ABB RAPID module: controlador3.mod

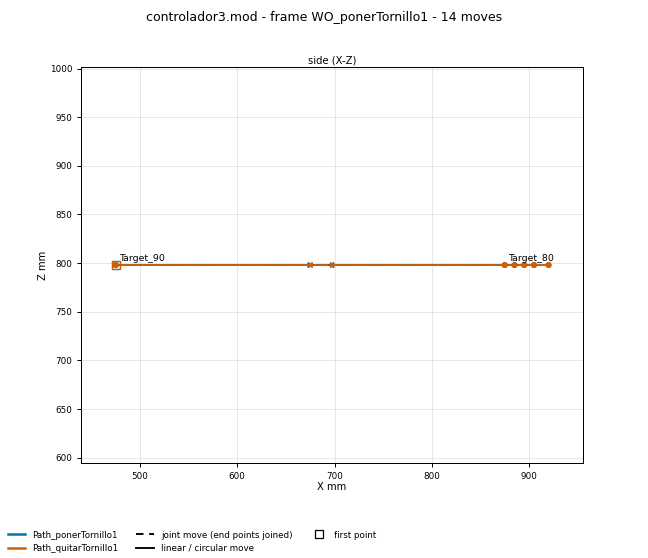
[picture p0: tool path of controlador3.mod in frame WO_ponerTornillo1, 14 of 120 moves have a stored position in this frame; points joined in program order, loops and branches not executed]
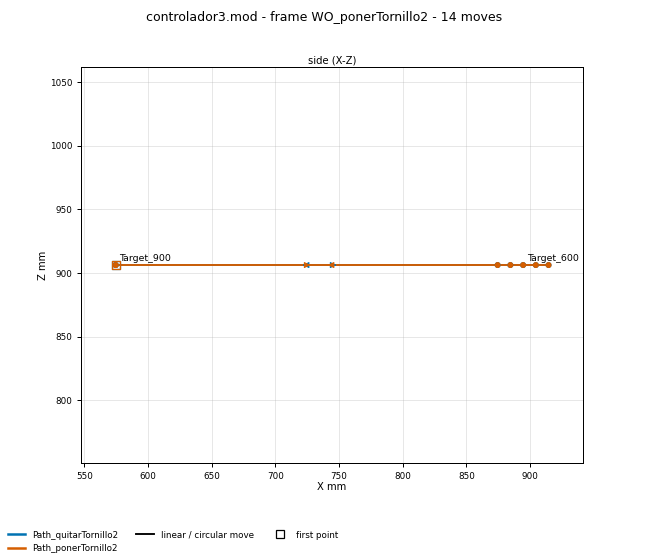
[picture p1: tool path of controlador3.mod in frame WO_ponerTornillo2, 14 of 120 moves have a stored position in this frame; points joined in program order, loops and branches not executed]
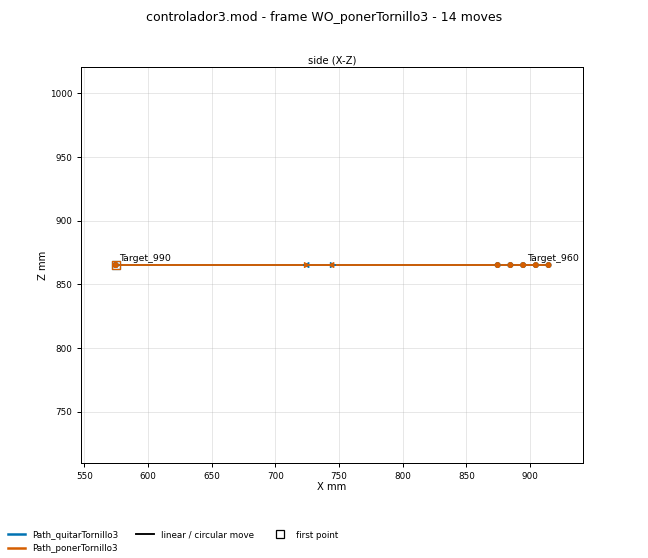
[picture p2: tool path of controlador3.mod in frame WO_ponerTornillo3, 14 of 120 moves have a stored position in this frame; points joined in program order, loops and branches not executed]
MODULE Module1
        CONST robtarget Target_30:=[[-0.058,698.771,342.903],[0,0,1,0],[1,0,1,0],[9E+09,9E+09,9E+09,9E+09,9E+09,9E+09]];
    CONST robtarget Target_20:=[[-0.058,698.771,142.903],[0,0,1,0],[1,0,1,0],[9E+09,9E+09,9E+09,9E+09,9E+09,9E+09]];
    CONST robtarget Target_10:=[[-0.058,698.771,57.903],[0,0,1,0],[0,0,0,0],[9E+09,9E+09,9E+09,9E+09,9E+09,9E+09]];
    CONST robtarget Target_40:=[[920,-282.5,798],[0.707106781,0,0.707106781,0],[-1,1,-2,0],[9E+09,9E+09,9E+09,9E+09,9E+09,9E+09]];
    CONST robtarget Target_90:=[[475,-282.5,798],[0,0.707106781,0,0.707106781],[-1,1,0,0],[9E+09,9E+09,9E+09,9E+09,9E+09,9E+09]];
    CONST robtarget Target_80:=[[875,-282.5,798],[0,0.707106781,0,0.707106781],[-1,1,0,0],[9E+09,9E+09,9E+09,9E+09,9E+09,9E+09]];
    CONST robtarget Target_70:=[[885,-282.5,798],[0.27059805,-0.653281482,0.27059805,-0.653281482],[-1,1,1,0],[9E+09,9E+09,9E+09,9E+09,9E+09,9E+09]];
    CONST robtarget Target_60:=[[895,-282.5,798],[0.5,-0.5,0.5,-0.5],[-1,1,1,0],[9E+09,9E+09,9E+09,9E+09,9E+09,9E+09]];
    CONST robtarget Target_50:=[[905,-282.5,798],[0.62578076,-0.329239185,0.62578076,-0.329239185],[-1,1,-2,0],[9E+09,9E+09,9E+09,9E+09,9E+09,9E+09]];
    CONST robtarget Target_40_1:=[[910,-282.5,798],[0.694697338,-0.131892411,0.694697338,-0.131892411],[-1,1,-2,0],[9E+09,9E+09,9E+09,9E+09,9E+09,9E+09]];
    CONST robtarget Target_55:=[[905,-282.5,798],[0.653281482,-0.27059805,0.653281482,-0.27059805],[-1,1,-2,0],[9E+09,9E+09,9E+09,9E+09,9E+09,9E+09]];
    CONST robtarget Target_45:=[[915,-282.5,798],[0.707106781,0,0.707106781,0],[-1,1,-2,0],[9E+09,9E+09,9E+09,9E+09,9E+09,9E+09]];
    CONST robtarget Target_56:=[[900,-282.5,798],[0.587937801,-0.392847479,0.587937801,-0.392847479],[-1,1,1,0],[9E+09,9E+09,9E+09,9E+09,9E+09,9E+09]];
    CONST robtarget Target_300:=[[0.2,748.407,342.618],[0,0,1,0],[0,0,0,0],[9E+09,9E+09,9E+09,9E+09,9E+09,9E+09]];
    CONST robtarget Target_200:=[[0.2,748.407,142.618],[0,0,1,0],[0,0,0,0],[9E+09,9E+09,9E+09,9E+09,9E+09,9E+09]];
    CONST robtarget Target_100:=[[0.2,748.407,57.618],[0,0,1,0],[0,0,0,0],[9E+09,9E+09,9E+09,9E+09,9E+09,9E+09]];
    CONST robtarget Target_330:=[[0.975,798.745,343.167],[0,0,1,0],[0,0,0,0],[9E+09,9E+09,9E+09,9E+09,9E+09,9E+09]];
    CONST robtarget Target_320:=[[0.975,798.745,143.167],[0,0,1,0],[0,0,0,0],[9E+09,9E+09,9E+09,9E+09,9E+09,9E+09]];
    CONST robtarget Target_310:=[[0.975,798.745,57.167],[0,0,1,0],[0,0,0,0],[9E+09,9E+09,9E+09,9E+09,9E+09,9E+09]];
    CONST robtarget Target_360:=[[0.487,848.79,342.715],[0,0,1,0],[0,0,0,0],[9E+09,9E+09,9E+09,9E+09,9E+09,9E+09]];
    CONST robtarget Target_350:=[[0.487,848.79,142.715],[0,0,1,0],[0,0,0,0],[9E+09,9E+09,9E+09,9E+09,9E+09,9E+09]];
    CONST robtarget Target_340:=[[0.487,848.79,56.715],[0,0,1,0],[0,0,0,0],[9E+09,9E+09,9E+09,9E+09,9E+09,9E+09]];
    CONST robtarget Target_390:=[[0.244,898.683,343.055],[0,0,1,0],[0,0,0,0],[9E+09,9E+09,9E+09,9E+09,9E+09,9E+09]];
    CONST robtarget Target_380:=[[0.244,898.683,143.055],[0,0,1,0],[0,0,0,0],[9E+09,9E+09,9E+09,9E+09,9E+09,9E+09]];
    CONST robtarget Target_370:=[[0.244,898.683,57.055],[0,0,1,0],[0,0,0,0],[9E+09,9E+09,9E+09,9E+09,9E+09,9E+09]];
    CONST robtarget Target_900:=[[574.529,-360.533,906.323],[0,0.707106781,0,0.707106781],[0,0,0,0],[9E+09,9E+09,9E+09,9E+09,9E+09,9E+09]];
    CONST robtarget Target_400:=[[914.529,-360.533,906.323],[0.707106781,0,0.707106781,0],[-1,1,-2,0],[9E+09,9E+09,9E+09,9E+09,9E+09,9E+09]];
    CONST robtarget Target_500:=[[904.529,-360.533,906.323],[0.653281482,-0.27059805,0.653281482,-0.27059805],[-1,1,-2,0],[9E+09,9E+09,9E+09,9E+09,9E+09,9E+09]];
    CONST robtarget Target_600:=[[894.529,-360.533,906.323],[0.5,-0.5,0.5,-0.5],[-1,1,1,0],[9E+09,9E+09,9E+09,9E+09,9E+09,9E+09]];
    CONST robtarget Target_700:=[[884.529,-360.533,906.323],[0.27059805,-0.653281482,0.27059805,-0.653281482],[-1,1,1,0],[9E+09,9E+09,9E+09,9E+09,9E+09,9E+09]];
    CONST robtarget Target_800:=[[874.529,-360.533,906.323],[0,0.707106781,0,0.707106781],[-1,1,0,0],[9E+09,9E+09,9E+09,9E+09,9E+09,9E+09]];
    CONST robtarget Target_990:=[[574.529,-487.2,865.271],[0,0.707106781,0,0.707106781],[0,0,0,0],[9E+09,9E+09,9E+09,9E+09,9E+09,9E+09]];
    CONST robtarget Target_940:=[[914.529,-487.2,865.271],[0.707106781,0,0.707106781,0],[-1,1,-2,0],[9E+09,9E+09,9E+09,9E+09,9E+09,9E+09]];
    CONST robtarget Target_950:=[[904.529,-487.2,865.271],[0.653281482,-0.27059805,0.653281482,-0.27059805],[-1,1,-2,0],[9E+09,9E+09,9E+09,9E+09,9E+09,9E+09]];
    CONST robtarget Target_960:=[[894.529,-487.2,865.271],[0.5,-0.5,0.5,-0.5],[-1,1,1,0],[9E+09,9E+09,9E+09,9E+09,9E+09,9E+09]];
    CONST robtarget Target_970:=[[884.529,-487.2,865.271],[0.27059805,-0.653281482,0.27059805,-0.653281482],[-1,1,1,0],[9E+09,9E+09,9E+09,9E+09,9E+09,9E+09]];
    CONST robtarget Target_980:=[[874.529,-487.2,865.271],[0,0.707106781,0,0.707106781],[-1,1,0,0],[9E+09,9E+09,9E+09,9E+09,9E+09,9E+09]];
    CONST robtarget Target_9000:=[[574.029,-487.592,731.451],[0,0.707106781,0,0.707106781],[0,0,0,0],[9E+09,9E+09,9E+09,9E+09,9E+09,9E+09]];
    CONST robtarget Target_4000:=[[914.029,-487.592,731.451],[0.707106781,0,0.707106781,0],[-1,1,-2,0],[9E+09,9E+09,9E+09,9E+09,9E+09,9E+09]];
    CONST robtarget Target_5000:=[[904.029,-487.592,731.451],[0.653281482,-0.27059805,0.653281482,-0.27059805],[-1,1,-2,0],[9E+09,9E+09,9E+09,9E+09,9E+09,9E+09]];
    CONST robtarget Target_6000:=[[894.029,-487.592,731.451],[0.5,-0.5,0.5,-0.5],[-1,1,1,0],[9E+09,9E+09,9E+09,9E+09,9E+09,9E+09]];
    CONST robtarget Target_7000:=[[884.029,-487.592,731.451],[0.27059805,-0.653281482,0.27059805,-0.653281482],[-1,1,1,0],[9E+09,9E+09,9E+09,9E+09,9E+09,9E+09]];
    CONST robtarget Target_8000:=[[874.029,-487.592,731.451],[0,0.707106781,0,0.707106781],[-1,1,0,0],[9E+09,9E+09,9E+09,9E+09,9E+09,9E+09]];
    CONST robtarget Target_9090:=[[574.029,-360.611,690.519],[0,0.707106781,0,0.707106781],[0,0,0,0],[9E+09,9E+09,9E+09,9E+09,9E+09,9E+09]];
    CONST robtarget Target_9040:=[[914.029,-360.611,690.519],[0.707106781,0,0.707106781,0],[-1,1,-2,0],[9E+09,9E+09,9E+09,9E+09,9E+09,9E+09]];
    CONST robtarget Target_9050:=[[904.029,-360.611,690.519],[0.653281482,-0.27059805,0.653281482,-0.27059805],[-1,1,1,0],[9E+09,9E+09,9E+09,9E+09,9E+09,9E+09]];
    CONST robtarget Target_9060:=[[894.029,-360.611,690.519],[0.5,-0.5,0.5,-0.5],[-1,1,1,0],[9E+09,9E+09,9E+09,9E+09,9E+09,9E+09]];
    CONST robtarget Target_9070:=[[884.029,-360.611,690.519],[0.27059805,-0.653281482,0.27059805,-0.653281482],[-1,1,0,0],[9E+09,9E+09,9E+09,9E+09,9E+09,9E+09]];
    CONST robtarget Target_9080:=[[874.029,-360.611,690.519],[0,0.707106781,0,0.707106781],[-1,1,0,0],[9E+09,9E+09,9E+09,9E+09,9E+09,9E+09]];
!***********************************************************
    !
    ! Módulo:  Module1
    !
    ! Descripción:
    !   <Introduzca la descripción aquí>
    !
    ! Autor: KTCHIA
    !
    ! Versión: 1.0
    !
    !***********************************************************


    !***********************************************************
    !
    ! Procedimiento Main
    !
    !   Este es el punto de entrada de su programa
    !
    !***********************************************************
    PROC main()
        !Añada aquí su código}
        SetDO Q_finish,0;
        IF E_begin=0 THEN
            WaitDI E_begin,1;
        ENDIF
        IF E_begin = 1 THEN
            SetDO Q_gripper,0;
            Path_recogerTornillo1;
            Path_ponerTornillo1;
            Path_recogerTornillo2;
            Path_ponerTornillo2;
            Path_recogerTornillo3;
            Path_ponerTornillo3;
            Path_recogerTornillo4;
            Path_ponerTornillo4;
            Path_recogerTornillo5;
            Path_ponerTornillo5;
            Path_quitarTornillo1;
            Path_descargarTornillo1;
            Path_quitarTornillo2;
            Path_descargarTornillo2;
            Path_quitarTornillo3;
            Path_descargarTornillo3;
            Path_quitarTornillo4;
            Path_descargarTornillo4;
            Path_quitarTornillo5;
            Path_descargarTornillo5;
            SetDO Q_finish,1;
        ENDIF
    ENDPROC

    PROC Path_recogerTornillo1()
        MoveJ Target_30,v500,fine,Servo\WObj:=WO_cogerTornillo1;
        SetDO Q_gripper,0;
        WaitTime 1;
        MoveL Target_20,v500,fine,Servo\WObj:=WO_cogerTornillo1;
        MoveL Target_10,v500,fine,Servo\WObj:=WO_cogerTornillo1;
        SetDO Q_gripper,1;
        WaitTime 1;
        MoveL Target_20,v500,fine,Servo\WObj:=WO_cogerTornillo1;
        MoveL Target_30,v500,fine,Servo\WObj:=WO_cogerTornillo1;
    ENDPROC
    PROC Path_ponerTornillo1()
        MoveJ Target_90,v500,fine,Servo\WObj:=WO_ponerTornillo1;
        MoveL Target_80,v500,fine,Servo\WObj:=WO_ponerTornillo1;
        MoveL Target_70,v500,fine,Servo\WObj:=WO_ponerTornillo1;
        MoveJ Target_60,v500,fine,Servo\WObj:=WO_ponerTornillo1;
        SetDO Q_gripper,0;
        WaitTime 1;
        MoveJ Target_50,v500,fine,Servo\WObj:=WO_ponerTornillo1;
        SetDO Q_gripper,1;
        WaitTime 1;
        MoveJ Target_40,v500,fine,Servo\WObj:=WO_ponerTornillo1;
        SetDO Q_gripper,0;
        WaitTime 1;
        MoveL Target_90,v500,fine,Servo\WObj:=WO_ponerTornillo1;
    ENDPROC
    PROC Path_quitarTornillo1()
        MoveJ Target_90,v500,fine,Servo\WObj:=WO_ponerTornillo1;
        MoveL Target_40,v500,fine,Servo\WObj:=WO_ponerTornillo1;
        SetDO Q_gripper,1;
        WaitTime 1;
        MoveJ Target_50,v500,fine,Servo\WObj:=WO_ponerTornillo1;
        SetDO Q_gripper,0;
        WaitTime 1;
        MoveJ Target_60,v500,fine,Servo\WObj:=WO_ponerTornillo1;
        SetDO Q_gripper,1;
        WaitTime 1;
        MoveL Target_70,v500,fine,Servo\WObj:=WO_ponerTornillo1;
        MoveL Target_80,v500,fine,Servo\WObj:=WO_ponerTornillo1;
        MoveJ Target_90,v500,fine,Servo\WObj:=WO_ponerTornillo1;
    ENDPROC
    PROC Path_descargarTornillo1()
        MoveJ Target_30,v500,fine,Servo\WObj:=WO_cogerTornillo1;
        MoveL Target_20,v500,fine,Servo\WObj:=WO_cogerTornillo1;
        MoveL Target_10,v500,fine,Servo\WObj:=WO_cogerTornillo1;
        SetDO Q_gripper,0;
        WaitTime 1;
        MoveL Target_20,v500,fine,Servo\WObj:=WO_cogerTornillo1;
        MoveL Target_30,v500,fine,Servo\WObj:=WO_cogerTornillo1;
    ENDPROC
    PROC Path_recogerTornillo2()
        SetDO Q_gripper,0;
        MoveJ Target_300,v500,fine,Servo\WObj:=WO_cogerTornillo2;
        WaitTime 1;
        MoveL Target_200,v500,fine,Servo\WObj:=WO_cogerTornillo2;
        MoveL Target_100,v500,fine,Servo\WObj:=WO_cogerTornillo2;
        SetDO Q_gripper,1;
        WaitTime 3;
        MoveL Target_200,v500,fine,Servo\WObj:=WO_cogerTornillo2;
        MoveL Target_300,v500,fine,Servo\WObj:=WO_cogerTornillo2;
    ENDPROC
    PROC Path_recogerTornillo3()
        MoveJ Target_330,v500,fine,Servo\WObj:=WO_cogerTornillo3;
        SetDO Q_gripper,0;
        WaitTime 1;
        MoveL Target_320,v500,fine,Servo\WObj:=WO_cogerTornillo3;
        MoveL Target_310,v500,fine,Servo\WObj:=WO_cogerTornillo3;
        SetDO Q_gripper,1;
        WaitTime 1;
        MoveL Target_320,v500,fine,Servo\WObj:=WO_cogerTornillo3;
        MoveL Target_330,v500,fine,Servo\WObj:=WO_cogerTornillo3;
    ENDPROC
    PROC Path_recogerTornillo4()
        MoveJ Target_360,v500,fine,Servo\WObj:=WO_cogerTornillo4;
        SetDO Q_gripper,0;
        WaitTime 1;
        MoveL Target_350,v500,fine,Servo\WObj:=WO_cogerTornillo4;
        MoveL Target_340,v500,fine,Servo\WObj:=WO_cogerTornillo4;
        SetDO Q_gripper,1;
        WaitTime 1;
        MoveL Target_350,v500,fine,Servo\WObj:=WO_cogerTornillo4;
        MoveL Target_360,v500,fine,Servo\WObj:=WO_cogerTornillo4;
    ENDPROC
    PROC Path_recogerTornillo5()
        MoveJ Target_390,v500,fine,Servo\WObj:=WO_cogerTornillo5;
        SetDO Q_gripper,0;
        WaitTime 1;
        MoveL Target_380,v500,fine,Servo\WObj:=WO_cogerTornillo5;
        MoveL Target_370,v500,fine,Servo\WObj:=WO_cogerTornillo5;
        SetDO Q_gripper,1;
        WaitTime 1;
        MoveL Target_380,v500,fine,Servo\WObj:=WO_cogerTornillo5;
        MoveL Target_390,v500,fine,Servo\WObj:=WO_cogerTornillo5;
    ENDPROC
    PROC Path_quitarTornillo2()
        MoveJ Target_900,v500,fine,Servo\WObj:=WO_ponerTornillo2;
        MoveL Target_400,v500,fine,Servo\WObj:=WO_ponerTornillo2;
        SetDO Q_gripper,1;
        WaitTime 1;
        MoveL Target_500,v500,fine,Servo\WObj:=WO_ponerTornillo2;
        SetDO Q_gripper,0;
        WaitTime 1;
        MoveL Target_600,v500,fine,Servo\WObj:=WO_ponerTornillo2;
        SetDO Q_gripper,1;
        WaitTime 1;
        MoveL Target_700,v500,fine,Servo\WObj:=WO_ponerTornillo2;
        MoveL Target_800,v500,fine,Servo\WObj:=WO_ponerTornillo2;
        MoveL Target_900,v500,fine,Servo\WObj:=WO_ponerTornillo2;
    ENDPROC
    PROC Path_quitarTornillo3()
        MoveJ Target_990,v500,fine,Servo\WObj:=WO_ponerTornillo3;
        MoveL Target_940,v500,fine,Servo\WObj:=WO_ponerTornillo3;
        SetDO Q_gripper,1;
        WaitTime 1;
        MoveL Target_950,v500,fine,Servo\WObj:=WO_ponerTornillo3;
        SetDO Q_gripper,0;
        WaitTime 1;
        MoveL Target_960,v500,fine,Servo\WObj:=WO_ponerTornillo3;
        SetDO Q_gripper,1;
        WaitTime 1;
        MoveL Target_970,v500,fine,Servo\WObj:=WO_ponerTornillo3;
        MoveL Target_980,v500,fine,Servo\WObj:=WO_ponerTornillo3;
        MoveL Target_990,v500,fine,Servo\WObj:=WO_ponerTornillo3;
    ENDPROC
    PROC Path_quitarTornillo4()
        MoveJ Target_9000,v500,fine,Servo\WObj:=WO_ponerTornillo4;
        MoveL Target_4000,v500,fine,Servo\WObj:=WO_ponerTornillo4;
        SetDO Q_gripper,1;
        WaitTime 1;
        MoveL Target_5000,v500,fine,Servo\WObj:=WO_ponerTornillo4;
        SetDO Q_gripper,0;
        WaitTime 1;
        MoveL Target_6000,v500,fine,Servo\WObj:=WO_ponerTornillo4;
        SetDO Q_gripper,1;
        WaitTime 1;
        MoveL Target_7000,v500,fine,Servo\WObj:=WO_ponerTornillo4;
        MoveL Target_8000,v500,fine,Servo\WObj:=WO_ponerTornillo4;
        MoveL Target_9000,v500,fine,Servo\WObj:=WO_ponerTornillo4;
    ENDPROC
    PROC Path_quitarTornillo5()
        MoveJ Target_9090,v500,fine,Servo\WObj:=WO_ponerTornillo5;
        MoveL Target_9040,v500,fine,Servo\WObj:=WO_ponerTornillo5;
        SetDO Q_gripper,1;
        WaitTime 1;
        MoveL Target_9050,v500,fine,Servo\WObj:=WO_ponerTornillo5;
        SetDO Q_gripper,0;
        WaitTime 1;
        MoveL Target_9060,v500,fine,Servo\WObj:=WO_ponerTornillo5;
        SetDO Q_gripper,1;
        WaitTime 1;
        MoveL Target_9070,v500,fine,Servo\WObj:=WO_ponerTornillo5;
        MoveL Target_9080,v500,fine,Servo\WObj:=WO_ponerTornillo5;
        MoveL Target_9090,v500,fine,Servo\WObj:=WO_ponerTornillo5;
    ENDPROC
    PROC Path_ponerTornillo2()
        MoveJ Target_900,v500,fine,Servo\WObj:=WO_ponerTornillo2;
        MoveL Target_800,v500,fine,Servo\WObj:=WO_ponerTornillo2;
        MoveL Target_700,v500,fine,Servo\WObj:=WO_ponerTornillo2;
        MoveL Target_600,v500,fine,Servo\WObj:=WO_ponerTornillo2;
        SetDO Q_gripper,0;
        WaitTime 1;
        MoveL Target_500,v500,fine,Servo\WObj:=WO_ponerTornillo2;
        SetDO Q_gripper,1;
        WaitTime 1;
        MoveL Target_400,v500,fine,Servo\WObj:=WO_ponerTornillo2;
        SetDO Q_gripper,0;
        WaitTime 1;
        MoveL Target_900,v500,fine,Servo\WObj:=WO_ponerTornillo2;
    ENDPROC
    PROC Path_ponerTornillo3()
        MoveJ Target_990,v500,fine,Servo\WObj:=WO_ponerTornillo3;
        MoveL Target_980,v500,fine,Servo\WObj:=WO_ponerTornillo3;
        MoveL Target_970,v500,fine,Servo\WObj:=WO_ponerTornillo3;
        MoveL Target_960,v500,fine,Servo\WObj:=WO_ponerTornillo3;
        SetDO Q_gripper,0;
        WaitTime 1;
        MoveL Target_950,v500,fine,Servo\WObj:=WO_ponerTornillo3;
        SetDO Q_gripper,1;
        WaitTime 1;
        MoveL Target_940,v500,fine,Servo\WObj:=WO_ponerTornillo3;
        SetDO Q_gripper,0;
        WaitTime 1;
        MoveL Target_990,v500,fine,Servo\WObj:=WO_ponerTornillo3;
    ENDPROC
    PROC Path_ponerTornillo4()
        MoveJ Target_9000,v500,fine,Servo\WObj:=WO_ponerTornillo4;
        MoveL Target_8000,v500,fine,Servo\WObj:=WO_ponerTornillo4;
        MoveL Target_7000,v500,fine,Servo\WObj:=WO_ponerTornillo4;
        MoveL Target_6000,v500,fine,Servo\WObj:=WO_ponerTornillo4;
        SetDO Q_gripper,0;
        WaitTime 1;
        MoveL Target_5000,v500,fine,Servo\WObj:=WO_ponerTornillo4;
        SetDO Q_gripper,1;
        WaitTime 1;
        MoveL Target_4000,v500,fine,Servo\WObj:=WO_ponerTornillo4;
        SetDO Q_gripper,0;
        WaitTime 1;
        MoveL Target_9000,v500,fine,Servo\WObj:=WO_ponerTornillo4;
    ENDPROC
    PROC Path_ponerTornillo5()
        MoveJ Target_9090,v500,fine,Servo\WObj:=WO_ponerTornillo5;
        MoveL Target_9080,v500,fine,Servo\WObj:=WO_ponerTornillo5;
        MoveL Target_9070,v500,fine,Servo\WObj:=WO_ponerTornillo5;
        MoveL Target_9060,v500,fine,Servo\WObj:=WO_ponerTornillo5;
        SetDO Q_gripper,0;
        WaitTime 1;
        MoveL Target_9050,v500,fine,Servo\WObj:=WO_ponerTornillo5;
        SetDO Q_gripper,1;
        WaitTime 1;
        MoveL Target_9040,v500,fine,Servo\WObj:=WO_ponerTornillo5;
        SetDO Q_gripper,0;
        WaitTime 1;
        MoveL Target_9090,v500,fine,Servo\WObj:=WO_ponerTornillo5;
    ENDPROC
    PROC Path_descargarTornillo2()
        MoveJ Target_300,v500,fine,Servo\WObj:=WO_cogerTornillo2;
        MoveL Target_200,v500,fine,Servo\WObj:=WO_cogerTornillo2;
        MoveL Target_100,v500,fine,Servo\WObj:=WO_cogerTornillo2;
        SetDO Q_gripper,0;
        WaitTime 1;
        MoveL Target_200,v500,fine,Servo\WObj:=WO_cogerTornillo2;
        MoveL Target_300,v500,fine,Servo\WObj:=WO_cogerTornillo2;
    ENDPROC
    PROC Path_descargarTornillo3()
        MoveJ Target_330,v500,fine,Servo\WObj:=WO_cogerTornillo3;
        MoveL Target_320,v500,fine,Servo\WObj:=WO_cogerTornillo3;
        MoveL Target_310,v500,fine,Servo\WObj:=WO_cogerTornillo3;
        SetDO Q_gripper,0;
        WaitTime 1;
        MoveL Target_320,v500,fine,Servo\WObj:=WO_cogerTornillo3;
        MoveL Target_330,v500,fine,Servo\WObj:=WO_cogerTornillo3;
    ENDPROC
    PROC Path_descargarTornillo4()
        MoveJ Target_360,v500,fine,Servo\WObj:=WO_cogerTornillo4;
        MoveL Target_350,v500,fine,Servo\WObj:=WO_cogerTornillo4;
        MoveL Target_340,v500,fine,Servo\WObj:=WO_cogerTornillo4;
        SetDO Q_gripper,0;
        WaitTime 1;
        MoveL Target_350,v500,fine,Servo\WObj:=WO_cogerTornillo4;
        MoveL Target_360,v500,fine,Servo\WObj:=WO_cogerTornillo4;
    ENDPROC
    PROC Path_descargarTornillo5()
        MoveJ Target_390,v500,fine,Servo\WObj:=WO_cogerTornillo5;
        MoveL Target_380,v500,fine,Servo\WObj:=WO_cogerTornillo5;
        MoveL Target_370,v500,fine,Servo\WObj:=WO_cogerTornillo5;
        SetDO Q_gripper,0;
        WaitTime 1;
        MoveL Target_380,v500,fine,Servo\WObj:=WO_cogerTornillo5;
        MoveL Target_390,v500,fine,Servo\WObj:=WO_cogerTornillo5;
    ENDPROC
ENDMODULE
